(* IEC 61131-3 sources: volt/packages/volt-lsp-iec/test-corpus/pro2193/Device/Plc Logic/Application/09 Misc/Library Manager/(unresolved)/cmpiomgr interfaces, 17 files *)

(* ---- EVTPARAM_CMPIOMGR.dut ---- *)
TYPE EVTPARAM_CMPIOMGR :
STRUCT
	PCONNECTORLIST : POINTER TO IoConfigConnector;
	NCOUNT : DINT;
END_STRUCT
END_TYPE

(* ---- IOCONFIGCHANNELMAP.dut ---- *)
TYPE IOCONFIGCHANNELMAP :
STRUCT
	PPARAMETER : POINTER TO IoConfigParameter;
	PBYIECADDRESS : POINTER TO BYTE;
	WPARAMETERBITOFFSET : WORD;
	WIECADDRESSBITOFFSET : WORD;
	WSIZE : WORD;
	WDUMMY : WORD;
	DWDRIVERSPECIFIC : XWORD;
END_STRUCT
END_TYPE

(* ---- IOCONFIGCONNECTOR.dut ---- *)
TYPE IOCONFIGCONNECTOR :
STRUCT
	WTYPE : WORD;
	WOPTIONS : WORD;
	DWFLAGS : DWORD;
	HIODRV : RTS_IEC_HANDLE;
	DWNUMOFPARAMETERS : DWORD;
	PPARAMETERLIST : POINTER TO IoConfigParameter;
	PFATHER : POINTER TO IoConfigConnector;
END_STRUCT
END_TYPE

(* ---- IOCONFIGCONNECTORMAP.dut ---- *)
TYPE IOCONFIGCONNECTORMAP :
STRUCT
	PCONNECTOR : POINTER TO IoConfigConnector;
	DWIOMGRSPECIFIC : XWORD;
	DWNUMOFCHANNELS : DWORD;
	PCHANNELMAPLIST : POINTER TO IoConfigChannelMap;
END_STRUCT
END_TYPE

(* ---- IOCONFIGPARAMETER.dut ---- *)
TYPE IOCONFIGPARAMETER :
STRUCT
	DWPARAMETERID : DWORD;
	DWVALUE : XWORD;
	WTYPE : WORD;
	WLEN : WORD;
	DWFLAGS : DWORD;
	DWDRIVERSPECIFIC : XWORD;
END_STRUCT
END_TYPE

(* ---- IOCONFIGTASKMAP.dut ---- *)
TYPE IOCONFIGTASKMAP :
STRUCT
	DWTASKID : DWORD;
	WTYPE : WORD;
	WNUMOFCONNECTORMAP : WORD;
	PCONNECTORMAPLIST : POINTER TO IoConfigConnectorMap;
END_STRUCT
END_TYPE

(* ---- BASETYPEINFORMATION.gvl ---- *)
VAR_GLOBAL
	CMLBT_MASK : WORD := 16#FF;
	CMLBT_IS_SET : WORD := 16#100;
	CMLBT_ENABLE : WORD := 16#8000;
END_VAR

(* ---- BUSCYCLETYPE.gvl ---- *)
VAR_GLOBAL
	BCT_START : UDINT := 16#1;
	BCT_END : UDINT := 16#2;
END_VAR

(* ---- BUSINDEPENDENTPARAMETERIDS.gvl ---- *)
VAR_GLOBAL
	FIP_NETX_DEVICE : UDINT := 16#70000000;
	FIP_WATCHDOG : UDINT := 16#70000001;
	FIP_NETX_SLOT_NUMBER : UDINT := 16#70000002;
	FIP_NETX_CHANNEL_NUMBER : UDINT := 16#70000003;
	FIP_BUS_ON_TIMEOUT : UDINT := 16#70000004;
	FIP_DEVICENAME : UDINT := 16#70000010;
	FIP_DEVICEIDENTIFICATION_HASH : UDINT := 16#70000011;
	FIP_UPDATE_IO_IN_STOP : UDINT := 16#70000012;
	FIP_SAFETY_PROTOCOL : UDINT := 16#70000018;
	FIP_CONFIG_VERSION : UDINT := 16#70001000;
	FIP_NUMBER_OF_SAFETY_PROTOCOLS : UDINT := 16#7F000018;
	FIP_FIRST_SAFETY_PROTOCOL_PARAM : UDINT := 16#7F000019;
	FIP_LAST_SAFETY_PROTOCOL_PARAM : UDINT := 16#7F000118;
END_VAR

(* ---- CONNECTORFLAGS.gvl ---- *)
VAR_GLOBAL
	CF_ENABLE : WORD := 16#1;
	CF_DIAG_PROVIDER : WORD := 16#2;
	CF_DEVICE_ENABLED : WORD := 16#4;
	CF_DEMOLICENSE_ACTIVE : WORD := 16#8;
	CF_DRIVER_AVAILABLE : WORD := 16#10;
	CF_CONNECTOR_FOUND : WORD := 16#20;
	CF_CONNECTOR_CONFIGURED : WORD := 16#40;
	CF_CONNECTOR_ACTIVE : WORD := 16#80;
	CF_CONNECTOR_BUS_ERROR : WORD := 16#100;
	CF_CONNECTOR_ERROR : WORD := 16#200;
	CF_CONNECTOR_DIAGNOSTIC_AVAILABLE : WORD := 16#400;
	CF_CONNECTOR_PASSIVE : WORD := 16#800;
	CF_ERROR_CLEARED : WORD := 16#1000;
END_VAR

(* ---- CONNECTOROPTIONS.gvl ---- *)
VAR_GLOBAL
	CO_NONE : WORD := 16#0;
	CO_SCAN_PENDING_SUPPORTED : WORD := 16#1;
END_VAR

(* ---- CONNECTORTYPES.gvl ---- *)
VAR_GLOBAL
	CT_PROGRAMMABLE : WORD := 16#1000;
	CT_PARAMETRIZABLE : WORD := 16#2000;
	CT_CAN_BUS : WORD := 16#F;
	CT_CAN_MASTER : WORD := 16#10;
	CT_CAN_SLAVE : WORD := 16#11;
	CT_CAN_DEVICE : WORD := 16#12;
	CT_CANOPEN_SAFETY : WORD := 16#15;
	CT_J1939_MANAGER : WORD := 16#18;
	CT_J1939_ECU : WORD := 16#19;
	CT_CANOPEN_SAFETY_SLAVE : WORD := 16#1A;
	CT_PROFIBUS_MASTER : WORD := 16#20;
	CT_PROFIBUS_SLAVE : WORD := 16#21;
	CT_PROFIBUS_DEVICE : WORD := 16#22;
	CT_PROFIBUS_MOD_MASTER : WORD := 16#23;
	CT_PROFIBUS_MOD_SLAVE : WORD := 16#24;
	CT_DEVICENET_MASTER : WORD := 16#30;
	CT_DEVICENET_SLAVE : WORD := 16#31;
	CT_DEVICENET_DEVICE : WORD := 16#32;
	CT_ETHERCAT_MASTER : WORD := 16#40;
	CT_ETHERCAT_SLAVE : WORD := 16#41;
	CT_ETHERCAT_DEVICE : WORD := 16#42;
	CT_ENIP_SCANNER : WORD := 16#64;
	CT_ENIP_REMOTE_ADAPTER : WORD := 16#65;
	CT_PCI_MASTER : WORD := 16#100;
	CT_PCI_SLAVE : WORD := 16#101;
END_VAR

(* ---- DRIVERPROPERTYFLAGS.gvl ---- *)
VAR_GLOBAL
	DRVPROP_CONSISTENCY : DWORD := 16#1;
	DRVPROP_WATCHDOG : DWORD := 16#2;
	DRVPROP_REDUNDANCY : DWORD := 16#4;
	DRVPROP_ACTIVE : DWORD := 16#8;
	DRVPROP_ERROR_ACTIVE : DWORD := 16#10;
	DRVPROP_ERROR_PASSIVE : DWORD := 16#20;
	DRVPROP_BACKGROUND_GETDIAG : DWORD := 16#40;
	DRVPROP_NO_SYNC : DWORD := 16#80;
END_VAR

(* ---- EVENTIDS.gvl ---- *)
VAR_GLOBAL
	CMPID_CMPIOMGR : DWORD := 16#12;
	EVTPARAMID_CMPIOMGR : WORD := 16#1;
	EVTVERSION_CMPIOMGR : WORD := 16#1;
	EVT_PREPAREUPDATECONFIGURATION : DWORD := 16#10001;
	EVT_UPDATECONFIGURATIONDONE : DWORD := 16#10002;
	EVT_CONFIGAPPSTARTEDDONE : DWORD := 16#10003;
	EVT_PREPARECONFIGAPPSTOPPED : DWORD := 16#10004;
	EVT_CONFIGAPPSTOPPEDDONE : DWORD := 16#10008;
END_VAR

(* ---- LOCKSCOPES.gvl ---- *)
VAR_GLOBAL
	IOMGR_LOCK_READ_INPUTS : DWORD := 16#1;
	IOMGR_LOCK_WRITE_OUTPUTS : DWORD := 16#2;
END_VAR

(* ---- PARAMETERVALUEFLAGS.gvl ---- *)
VAR_GLOBAL
	PVF_FUNCTION : WORD := 16#1;
	PVF_POINTER : WORD := 16#2;
	PVF_VALUE : WORD := 16#4;
	PVF_READ : WORD := 16#10;
	PVF_WRITE : WORD := 16#20;
	PVF_BIDIRECTIONAL : WORD := 16#100;
END_VAR

(* ---- TASKMAPTYPES.gvl ---- *)
VAR_GLOBAL
	TMT_INPUTS : WORD := 16#1;
	TMT_OUTPUTS : WORD := 16#2;
END_VAR
